KUKA KRL program: chk_w5_wechs_ok.src

&ACCESS RVO2
&COMMENT Check Gripper Actros
DEF chk_w5_wechs_ok( )

; VERIFICAÇÃO DE FERRAMENTA: Gripper Actros

$TIMER[10] = 0
$TIMER_STOP[10] = FALSE

wait for (($in[161]) and ($in[169]) and ($in[177]) and ($IN[185]) and (not $IN[193]) and ($IN[201]) and ($IN[209]) and ($IN[219]))

$TIMER_STOP[10] = TRUE
$TIMER[10] = 0

;//---- End -------
;Diag_Appl(#Off,5)

END
